# EPICS autosave request: iocBoot/iocTomoScan_13BM_MCS/auto_settings.req
file "tomoScan_settings.req", P=$(P), R=$(R)
file "tomoScan_13BM_settings.req", P=$(P), R=$(R)
file "tomoScan_13BM_MCS_settings.req", P=$(P), R=$(R)
